// TIA Portal V19 export
TYPE "typeCanProcessImageInputs"
   STRUCT
      BufferA : Struct
         SlaveDigitalInput1 : Byte;
         SlaveDigitalInput2 : Byte;
         SlaveAnalogInput1 : Int;
         SlaveAnalogInput2 : Int;
         SlaveAnalogInput3 : Int;
         SlaveAnalogInput4 : Int;
      END_STRUCT;
      BufferB : Struct
         SlaveDigitalInput1 : Byte;
         SlaveDigitalInput2 : Byte;
         SlaveAnalogInput1 : Int;
         SlaveAnalogInput2 : Int;
         SlaveAnalogInput3 : Int;
         SlaveAnalogInput4 : Int;
      END_STRUCT;
      ActiveBuffer : Byte;   // 0 = BufferA, 1 = BufferB. ActiveBuffer is the buffer the PC reads from, and the inactive buffer is the buffer the PLC updates from the input CAN process image.
   END_STRUCT;
END_TYPE
